FUNCTION NoOfRunningPumps : INT
VAR_IN_OUT
	Pumps		:	ARRAY[1..GVL.MAX_PUMPS] OF PumpType;
END_VAR
VAR
	Idx			:	INT;
	No			:	INT:=0;	// counter of running pumps
END_VAR

(* 
Count number of running pumps
*)

FOR Idx:=1 TO GVL.MAX_PUMPS DO
	IF Pumps[Idx].RunState = PumpState.RUN THEN
		No:=No+1;
	END_IF
END_FOR

NoOfRunningPumps := No;

END_FUNCTION

(* stored: Version 1.1.0.1, ProductVersion 3.1.4024.15
   POU NoOfRunningPumps: Id {dd70382d-6e0f-470d-9426-b3c91619a8d5}, SpecialFunc None *)
